// TIA Portal project "TestNivel" (V15.1)

(* hardware
DEVICE "S7-1200 station_1"  S7-1200 Station
   slot 0: "Rack_0"  S7-1200 Rack  Rack  V1.0
   slot 1: "PLC_1"  CPU 1214C AC/DC/Rly  6ES7 214-1BG40-0XB0  V4.2
*)

// ===== PLC "PLC_1"  CPU 1214C AC/DC/Rly =====

VAR_GLOBAL   // PLC tag table "Tabla de variables estándar"
   "sensor_nivel_1" AT %I0.0 : Bool;
   "sensor_nivel_2" AT %I0.1 : Bool;
   "sensor_nivel_3" AT %I0.2 : Bool;
   "DIN2" AT %Q0.1 : Bool;
   "DIN3" AT %Q0.2 : Bool;
END_VAR

ORGANIZATION_BLOCK "Main"   // OB1, LAD, ProgramCycle
TITLE = "Main Program Sweep (Cycle)"
{ S7_Optimized_Access := 'TRUE' }
VERSION : 0.1
   VAR_INPUT
      Initial_Call : Bool;   // Initial call of this OB
      Remanence : Bool;   // =True, if remanent data are available
   END_VAR
BEGIN

REGION Network 1
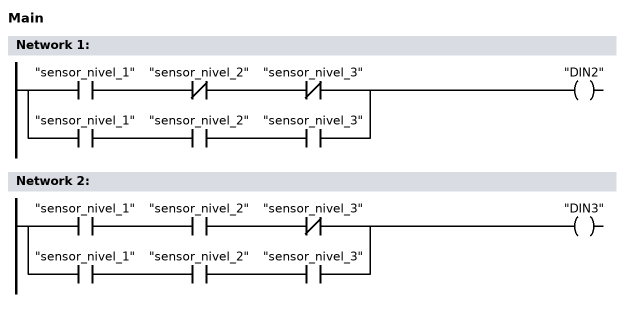
   RUNG wire#powerrail
      Contact( "sensor_nivel_1" )
      I_Contact( "sensor_nivel_2" )
      I_Contact( "sensor_nivel_3" )
      wire#w1
      Coil( "DIN2" )
   END_RUNG
   RUNG wire#powerrail
      Contact( "sensor_nivel_1" )
      Contact( "sensor_nivel_2" )
      Contact( "sensor_nivel_3" )
   END_RUNG wire#w1
   // the same network as SCL:
   "DIN2" := ("sensor_nivel_1" AND NOT "sensor_nivel_2" AND NOT "sensor_nivel_3") OR ("sensor_nivel_1" AND "sensor_nivel_2" AND "sensor_nivel_3");
END_REGION

REGION Network 2
   RUNG wire#powerrail
      Contact( "sensor_nivel_1" )
      Contact( "sensor_nivel_2" )
      I_Contact( "sensor_nivel_3" )
      wire#w1
      Coil( "DIN3" )
   END_RUNG
   RUNG wire#powerrail
      Contact( "sensor_nivel_1" )
      Contact( "sensor_nivel_2" )
      Contact( "sensor_nivel_3" )
   END_RUNG wire#w1
   // the same network as SCL:
   "DIN3" := ("sensor_nivel_1" AND "sensor_nivel_2" AND NOT "sensor_nivel_3") OR ("sensor_nivel_1" AND "sensor_nivel_2" AND "sensor_nivel_3");
END_REGION
END_ORGANIZATION_BLOCK